PROGRAM TimeStamp
VAR
	UnixTime: UnixTimestamp;
END_VAR

UnixTime(SyncTimeEnable := TRUE);

GVL_SW.Unix_TimeStamp := UnixTime.Milliseconds;

END_PROGRAM

(* stored: Version 1.1.0.1, ProductVersion 3.1.4024.15
   POU TimeStamp: Id {98a6470b-cf50-42d4-91f7-fb1ecaf72248}, SpecialFunc None *)
